# B&R Automation Studio project DeltaBot
Automation Studio 6.7.0.187; technology packages: mappCockpit 6.7.0, mappMotion 6.7.2, mappView 6.7.0, OpcUaCs 6.7.0

## Configuration X20EM0613

CPU X20EM0613, AutomationRuntime 6.7.8, Build 11.3.0

### Task classes (Cpu.sw)
```
Cyclic#4:
  Program <- Program.prg
Libraries: CoTrace, runtime, AsZip, FileIO, McBase, McAxis, MpRobotics, McAxGroup, McPathGen, McProgInt, McAcpAx, MpAxis, MpBase, McStpAx
```

### Hardware
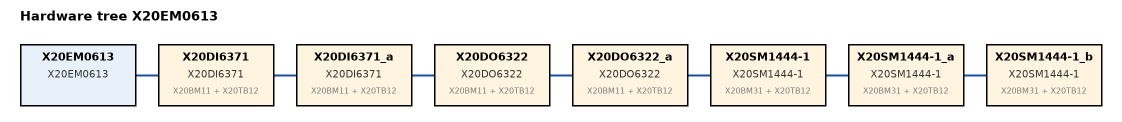
```
X20BM11 : X20BM11 v1.1.0.0  [X2X1 -> X20EM0613.IF6]
X20BM11_a : X20BM11 v1.1.0.0  [X2X1 -> X20BM11.X2X2]
X20BM11_b : X20BM11 v1.1.0.0  [X2X1 -> X20BM11_a.X2X2]
X20BM11_c : X20BM11 v1.1.0.0  [X2X1 -> X20BM11_b.X2X2]
X20BM31 : X20BM31 v1.1.0.0  [X2X1 -> X20BM11_c.X2X2]
X20BM31_a : X20BM31 v1.1.0.0  [X2X1 -> X20BM31.X2X2]
X20BM31_b : X20BM31 v1.1.0.0  [X2X1 -> X20BM31_a.X2X2]
X20DI6371 : X20DI6371 v1.3.0.0  [SS1 -> X20TB12_a.SS; SL -> X20BM11.SL1]
X20DI6371_a : X20DI6371 v1.3.0.0  [SS1 -> X20TB12_b.SS; SL -> X20BM11_a.SL1]
X20DO6322 : X20DO6322 v1.5.0.0  [SS1 -> X20TB12_c.SS; SL -> X20BM11_b.SL1]
X20DO6322_a : X20DO6322 v1.5.0.0  [SS1 -> X20TB12_d.SS; SL -> X20BM11_c.SL1]
X20EM0613 : X20EM0613 v1.1.1.0
  Connector IF2:
    ActivateDevice = 1
    Mode = Manual
    InternetAddress = 10.0.0.2
    SubnetMask = 255.255.255.0
    ActivateSnmp = 2
  ConfigurationID = DeltaBot_X20CP0484
  Simulation = 1
  TimerDeviceType = EPLX2X
  TimerDevice = X20EM0613.IF3
  TaskClassIdleTime = 4000
  Cyclic1Duration = 4000
  Cyclic1Tolerance = 0
  Cyclic1Output = 1
  Cyclic3Duration = 48000
  Cyclic3Tolerance = 48000
  Cyclic8Duration = 8000
  FileDevice1
  FileDeviceName1 = USER
  FileDevicePath1 = USER_PATH
X20SM1444-1 : X20SM1444-1 v3.0.0.0  [SS1 -> X20TB12_e.SS; SL -> X20BM31.SL1]
  FunctionModel/DriveConfiguration/Encoder/Encoder:
    InterfaceType = Incremental
  FunctionModel/DriveConfiguration/Encoder/Encoder/InterfaceType:
    LinesPerRevolution = 16384
  FunctionModel/DriveConfiguration/Channel[1]/RealAxis:
    AxisReference = gAxisQ1
  FunctionModel/DriveConfiguration/Channel[1]/RealAxis/MechanicalElements/RotaryToLinearTransformation:
    ReferenceDistance = 94.405
  FunctionModel/DriveConfiguration/Channel[1]/RealAxis:
    EncoderLink = OneEncoder
  FunctionModel/DriveConfiguration/Channel[1]/RealAxis/EncoderLink:
    PositionEncoder = Encoder
X20SM1444-1_a : X20SM1444-1 v3.0.0.0  [SS1 -> X20TB12_f.SS; SL -> X20BM31_a.SL1]
  FunctionModel/DriveConfiguration/Encoder/Encoder:
    InterfaceType = Incremental
  FunctionModel/DriveConfiguration/Encoder/Encoder/InterfaceType:
    LinesPerRevolution = 16384
  FunctionModel/DriveConfiguration/Channel[1]/RealAxis:
    AxisReference = gAxisQ2
  FunctionModel/DriveConfiguration/Channel[1]/RealAxis/MechanicalElements/RotaryToLinearTransformation:
    ReferenceDistance = 94.405
  FunctionModel/DriveConfiguration/Channel[1]/RealAxis:
    EncoderLink = OneEncoder
  FunctionModel/DriveConfiguration/Channel[1]/RealAxis/EncoderLink:
    PositionEncoder = Encoder
X20SM1444-1_b : X20SM1444-1 v3.0.0.0  [SS1 -> X20TB12_g.SS; SL -> X20BM31_b.SL1]
  FunctionModel/DriveConfiguration/Encoder/Encoder:
    InterfaceType = Incremental
  FunctionModel/DriveConfiguration/Encoder/Encoder/InterfaceType:
    LinesPerRevolution = 16384
  FunctionModel/DriveConfiguration/Channel[1]/RealAxis:
    AxisReference = gAxisQ3
  FunctionModel/DriveConfiguration/Channel[1]/RealAxis/MechanicalElements/RotaryToLinearTransformation:
    ReferenceDistance = 94.405
  FunctionModel/DriveConfiguration/Channel[1]/RealAxis:
    EncoderLink = OneEncoder
  FunctionModel/DriveConfiguration/Channel[1]/RealAxis/EncoderLink:
    PositionEncoder = Encoder
X20TB12_a : X20TB12 v1.0.0.0
X20TB12_b : X20TB12 v1.0.0.0
X20TB12_c : X20TB12 v1.0.0.0
X20TB12_d : X20TB12 v1.0.0.0
X20TB12_e : X20TB12 v1.0.0.0
X20TB12_f : X20TB12 v1.0.0.0
X20TB12_g : X20TB12 v1.0.0.0
```

### Config_1.axesgroup - X20EM0613/mappMotion/3AxesDeltaB/Config_1.axesgroup
```
Element g3AxDeltaB (Type=axesgroup)
  Type = PathGenAxesGroup
    PhysicalAxes:
      JointAxes:
        JointAxis[1]:
          AxisRef = gAxisQ1
        JointAxis[2]:
          AxisRef = gAxisQ2
        JointAxis[3]:
          AxisRef = gAxisQ3
    MechanicalSystem:
      MechSysRef = MechSys_3AxDeltaB
    AxesGroupFeatures:
      FeatureRef[1] = Feature_Programs
      FeatureRef[2] = Feature_Jogging
      FeatureRef[3] = Feature_HomingOrder
```

### Config_2.axis - X20EM0613/mappMotion/3AxesDeltaB/Config_2.axis
```
Element gAxisQ1 (Type=axis)
  BaseType = LinearBounded
  MovementLimits:
    Position:
      LowerLimit = 0
      UpperLimit = 270
    Velocity:
      Velocity = 1000
    Acceleration:
      Acceleration = 10000
    Deceleration:
      Deceleration = 10000
Element gAxisQ2 (Type=axis)
  BaseType = LinearBounded
  MovementLimits:
    Position:
      LowerLimit = 0
      UpperLimit = 270
    Velocity:
      Velocity = 1000
    Acceleration:
      Acceleration = 10000
    Deceleration:
      Deceleration = 10000
Element gAxisQ3 (Type=axis)
  BaseType = LinearBounded
  MovementLimits:
    Position:
      LowerLimit = 0
      UpperLimit = 270
    Velocity:
      Velocity = 1000
    Acceleration:
      Acceleration = 10000
    Deceleration:
      Deceleration = 10000
Element gAxisQ4 (Type=axis)
  BaseType = RotaryBounded
  MovementLimits:
    Velocity:
      Velocity = 10.0
    Acceleration:
      Acceleration = 50.0
    Deceleration:
      Deceleration = 50.0
```

### Config_3.mechanicalsystem - X20EM0613/mappMotion/3AxesDeltaB/Config_3.mechanicalsystem
```
Element MechSys_3AxDeltaB (Type=mechanicalsystem)
  Type = Delta
    Subtype = 3AxesDeltaB
      Description:
        Dimensions:
          BasePlatform:
            Center:
              Z = 797.14
            Arm1LinkPoint:
              Radius = 420.36
            Arm2LinkPoint:
              Angle = 120.0
              Radius = 420.36
            Arm3LinkPoint:
              Angle = 240.0
              Radius = 420.36
          Arms:
            Arm1:
              ArmLength = 500
              ArmOffset = -435
              ArmAngle = 45
            Arm2:
              ArmLength = 500
              ArmOffset = -435
              ArmAngle = 45
            Arm3:
              ArmLength = 500
              ArmOffset = -435
              ArmAngle = 45
          EndEffectorPlatform:
            Arm1LinkPoint:
              Radius = 46.27
            Arm2LinkPoint:
              Radius = 46.27
            Arm3LinkPoint:
              Radius = 46.27
            TranslationToFlange:
              Z = -6
        Offsets:
          JointAxis[1]
          JointAxis[2]
          JointAxis[3]
        CountDirections:
          JointAxis[1]
          JointAxis[2]
          JointAxis[3]
      JointAxesPositionLimits:
        JointAxis[1]
        JointAxis[2]
        JointAxis[3]
```

### Config_4.axesgroupfeature - X20EM0613/mappMotion/3AxesDeltaB/Config_4.axesgroupfeature
```
Element Feature_Programs (Type=axesgroupfeature)
Element Feature_Jogging (Type=axesgroupfeature)
  Type = Jogging
```

### Config_5.axesgroupfeature - X20EM0613/mappMotion/3AxesDeltaB/Config_5.axesgroupfeature
```
Element Feature_HomingOrder (Type=axesgroupfeature)
  Type = HomingOrder
    TogetherGroup[1]:
      AxisRef[1] = gAxisQ1
      AxisRef[2] = gAxisQ2
      AxisRef[3] = gAxisQ3
```

## Logical view

Binary libraries used (declarations not repeated): operator, runtime, AsIecCon, CoTrace 6.7.0, AsZip, FileIO, McBase 6.7.2, McAxis 6.7.2, MpRobotics 6.7.2, McAxGroup 6.7.2, McPathGen 6.7.2, McProgInt 6.7.2, McAcpAx 6.7.2, MpAxis 6.7.2, McStpAx 6.7.2, MpBase 6.8.0, AsOpcUac 6.7.0, AsOpcUas 6.7.0

### Global.var - Global variables
```iecst
VAR
	DAxis : MpDelta3Axis;
	DPara : MpDelta3AxisParType;
	W : LREAL;
	V : LREAL;
	U : LREAL;
END_VAR
```


### Program Logical/Program (IEC)

#### Variables.var
```iecst
VAR
	state : USINT := 0;
END_VAR
```

#### Main.st
```iecst
PROGRAM _INIT
	// reference na robotický systém
	DAxis.MpLink := ADR(g3AxDeltaB);
	// přiřazení parametrů
	DAxis.Parameters := ADR(DPara);
	// povolení plné rychlosti
	DAxis.Override := 100;
	// povolení funkčního bloku
	DAxis.Enable := TRUE ;
	// přiřazení výchozího pohybového programu
	//DPara.ProgramName := ’Home .st ’;
	// Provedeni funkčního bloku robota
	DAxis();
END_PROGRAM

PROGRAM _CYCLIC
	(* Insert code here *)
	CASE state OF
		0: // zapnutí napájení motorů
			IF DAxis.Active AND DAxis.Info.ReadyToPowerOn
				AND DAxis.Info.CommunicationReady THEN
				DAxis.Power := TRUE ;
				state := 1;
			END_IF ;
		1: // nalezení výchozích bodů
			IF DAxis.PowerOn AND NOT DAxis.IsHomed THEN
				DAxis.Home := TRUE ;
			END_IF ;
			IF DAxis.IsHomed THEN
				DAxis.Home := FALSE ;
				state := 2;
			END_IF ;
	END_CASE;

	U := DAxis.Info.JointAxisPosition[0];
	V := DAxis.Info.JointAxisPosition[1];
	W := DAxis.Info.JointAxisPosition[2];

	DAxis();
END_PROGRAM

PROGRAM _EXIT
	(* Insert code here *)
	DAxis.Power := FALSE ;
	DAxis.Home := FALSE ;
	DAxis.MoveDirect := FALSE ;
	DAxis.MoveLinear := FALSE ;
	DAxis.MoveProgram := FALSE ;
	DAxis.Enable := FALSE ;
	// provedeni funkčního bloku robota
	DAxis();
END_PROGRAM
```

- Visualisation Logical/mappView (not shown)

Listed in the project but not available here: Logical/Global.typ
